PROGRAM MAIN
VAR
	iAlive : INT;
	Kat : BOOL;
	Hund : bool;
END_VAR

iALive := iAlive + 1;

END_PROGRAM

(* stored: Version 1.1.0.1
   POU MAIN: Id {fe1eaf0d-cea0-4d8d-a0ff-878a06b7d758}, SpecialFunc None *)
